TEXTLIST ToolNumber
  1 = 'laser'
  2 = 'screw'
  3 = 'demo'
  4 = 'lens'
  5 = 'spare'
   = ''
END_TEXTLIST

(* stored: Version 1.1.0.1, ProductVersion 3.1.4024.10
   TextList ToolNumber: Id {98c618f3-8ba4-4b0d-a522-a6ce0977db43} *)
